INTERFACE I_ShutDown

METHOD ShutDown : BOOL
VAR_INPUT
		GvlIdentifier : STRING;
END_VAR
END_METHOD

END_INTERFACE

(* stored: Version 1.1.0.1, ProductVersion 3.1.4024.6
   Itf I_ShutDown: Id {a35ad707-20a3-44ac-a565-a79de4fc6be3}
   Method ShutDown: Id {bff6cd5a-1b39-4fe3-9da8-f1c1563e03a0} *)
